FUNCTION F_IsAtPositionJoint : BOOL
VAR_IN_OUT
  actual : ARRAY[*] OF LREAL;
  target : ARRAY[*] OF LREAL;
  delta  : ARRAY[*] OF LREAL;
END_VAR
VAR
  actLower, actUpper : DINT;
  ind : DINT;
END_VAR

actLower := LOWER_BOUND(actual, 1);
actUpper := UPPER_BOUND(actual, 1); 

IF actLower > LOWER_BOUND(target,1) OR actLower > LOWER_BOUND(delta, 1) THEN
  F_LogWarning('actLower > LOWER_BOUND(target,1) OR actLower > LOWER_BOUND(delta, 1)');
  RETURN;
  
END_IF

IF actUpper > UPPER_BOUND(target,1) OR actLower > UPPER_BOUND(delta, 1) THEN
  F_LogWarning('actUpper > UPPER_BOUND(target,1) OR actLower > UPPER_BOUND(delta, 1)');
  RETURN;
  
END_IF

FOR ind := actLower TO actUpper DO
  F_IsAtPositionJoint := ABS(actual[ind] - target[ind]) < delta[ind];
  
  IF NOT F_IsAtPositionJoint THEN
    // any failure means not in position.
    RETURN;
    
	END_IF
  
END_FOR

END_FUNCTION

(* stored: Version 1.1.0.1
   POU F_IsAtPositionJoint: Id {d6526da3-44cd-40c3-9114-958574579872}, SpecialFunc None *)
